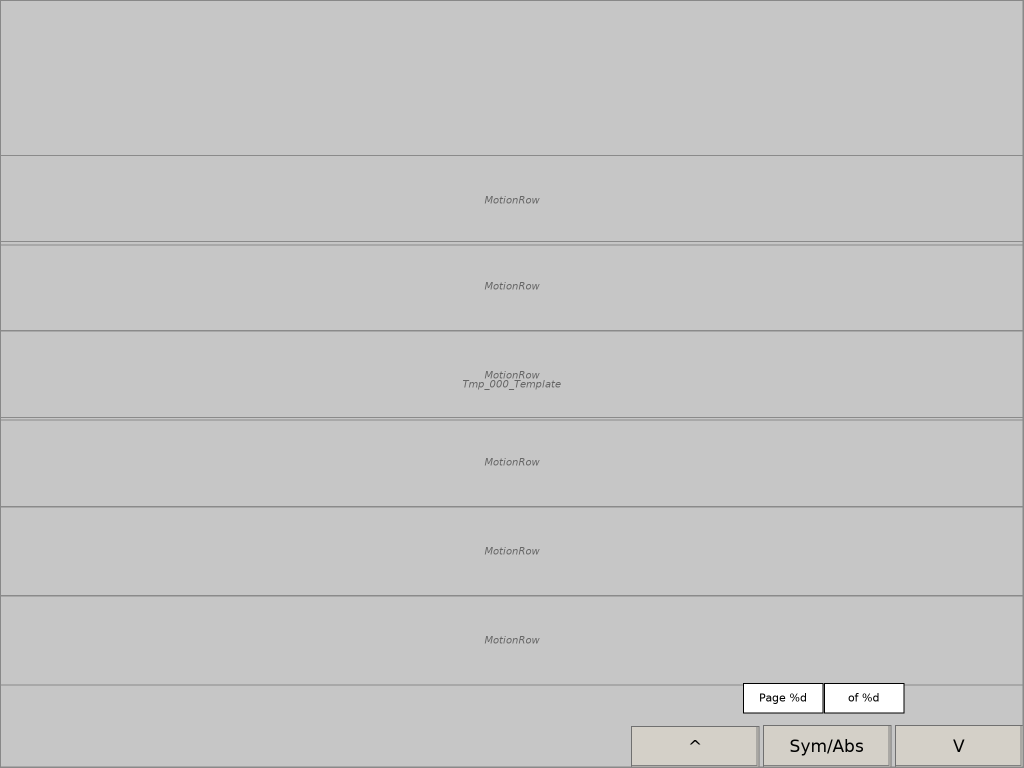
VISUALIZATION Mot_010_Motions  // 1024x768
    Frame (0,0 1024x768)
        shows Tmp_000_Template(header := gHMIData.hmiHeader)
    Frame (0,155 1024x90)
        shows MotionRow(MotionRowInstanceSingle := gHMIMotionRows.gMotionRows.gMotionRow1, MotionRowButtonsSingle := gHMIMotionRows.gMotionRowButtons.gMotionRow1btn)
    Frame (0,241 1024x90)
        shows MotionRow(MotionRowInstanceSingle := gHMIMotionRows.gMotionRows.gMotionRow2, MotionRowButtonsSingle := gHMIMotionRows.gMotionRowButtons.gMotionRow2btn)
    Frame (0,330 1024x90)
        shows MotionRow(MotionRowInstanceSingle := gHMIMotionRows.gMotionRows.gMotionRow3, MotionRowButtonsSingle := gHMIMotionRows.gMotionRowButtons.gMotionRow3btn)
    Frame (0,417 1024x90)
        shows MotionRow(MotionRowInstanceSingle := gHMIMotionRows.gMotionRows.gMotionRow4, MotionRowButtonsSingle := gHMIMotionRows.gMotionRowButtons.gMotionRow4btn)
    Frame (0,506 1024x90)
        shows MotionRow(MotionRowInstanceSingle := gHMIMotionRows.gMotionRows.gMotionRow5, MotionRowButtonsSingle := gHMIMotionRows.gMotionRowButtons.gMotionRow5btn)
    Frame (0,595 1024x90)
        shows MotionRow(MotionRowInstanceSingle := gHMIMotionRows.gMotionRows.gMotionRow6, MotionRowButtonsSingle := gHMIMotionRows.gMotionRowButtons.gMotionRow6btn)
    Button (763,725 128x42), "Sym/Abs", colour toggle: gHMIButtons.btnAbsMode
        toggle gHMIButtons.btnAbsMode
    Button (631,726 128x41), "^"
        tap gHMIButtons.btnPrevPage
    Button (895,725 128x42), "V"
        tap gHMIButtons.btnNextPage
    Rectangle (743,683 80x30), "Page %d", text variable: gHMIData.gActivePageNumber
    Rectangle (824,683 80x30), "of %d", text variable: gHMIData.gMaxPageNumber
END_VISUALIZATION

(* stored: Version 1.1.0.1, ProductVersion 3.1.4024.12
   Visu Mot_010_Motions: Id {6aba56b7-c6a1-4d88-88c9-c63feb9f8e06} *)
